TYPE ST_CartUIData :
STRUCT
	m_ergonomicCrl: ST_Ergonomic_control;
	m_cmdErgonomicCrl : ST_ergonomic_data;
	m_cmdCancelErgonPos :Vec4d;
	m_cmdJntPos :Vec4d;
END_STRUCT
END_TYPE

(* stored: Version 1.1.0.1, ProductVersion 3.1.4024.11
   DUT ST_CartUIData: Id {a5913571-fedf-4b0c-959b-43a014791c8b} *)
